FUNCTION_BLOCK FB_Statistic
VAR PERSISTENT
	bSaved:BOOL;
	Data:STRUCT_StatisticsData;
	DataSaved:STRUCT_StatisticsData;
	udiSamplesToSave:UDINT:=500;
	udiSamplesCounter:UDINT:=0;
END_VAR
VAR_INPUT
	bReset:BOOL;
	bRestore:BOOL;
END_VAR
VAR_OUTPUT
	rZScore:REAL;
END_VAR
VAR
	rValue:REAL;
END_VAR

METHOD PRIVATE M_calc_coef
VAR
	rCounter:REAL;
END_VAR
// Check counter and cast to real
IF THIS^.Data.udiCounter=0 THEN
	rCounter:=1;
END_IF
rCounter:=UDINT_TO_REAL(THIS^.Data.udiCounter);
// CALCULATE
// =======================================================
THIS^.Data.rStatCoef:=MAX((1/rCounter),THIS^.Data.rStatCoefMin);
// =======================================================
END_METHOD

METHOD PRIVATE M_calc_dev
VAR
	rRes:REAL;
END_VAR
IF THIS^.Data.rStatCoef=0 OR THIS^.Data.rStatCoef=1 THEN
	THIS^.Data.rDevSum:=0;
ELSE
	IF (THIS^.rValue-THIS^.Data.rMean)=0 THEN
		rRes:=0;
	ELSE
		rRes:=EXPT(THIS^.rValue-THIS^.Data.rMean,2);
	END_IF
	THIS^.Data.rDevSum :=	((1-THIS^.Data.rStatCoef)*THIS^.Data.rDevSum) + 
							(THIS^.Data.rStatCoef*rRes);
END_IF

IF THIS^.Data.rDevSum=0 THEN
	THIS^.Data.rDev:=0;
ELSE
	THIS^.Data.rDev:=SQRT(THIS^.Data.rDevSum);
END_IF
END_METHOD

METHOD PRIVATE M_calc_mean
VAR_INPUT
END_VAR
IF THIS^.Data.rStatCoef=1 THEN
	THIS^.Data.rMean:=THIS^.rValue;
ELSE
	IF THIS^.Data.rStatCoef<>0 THEN
		THIS^.Data.rMean := ((1-THIS^.Data.rStatCoef)*THIS^.Data.rMean) + 
							(THIS^.Data.rStatCoef*THIS^.rValue);
	end_if
END_IF
END_METHOD

METHOD PRIVATE M_calc_min_max
IF THIS^.Data.udiCounter=1 THEN
	THIS^.Data.rMaximum:=THIS^.rValue;
	THIS^.Data.rMinimum:=THIS^.rValue;
END_IF
THIS^.Data.rMinimum:=MIN(THIS^.Data.rMinimum,THIS^.rValue);
THIS^.Data.rMaximum:=MAX(THIS^.Data.rMaximum,THIS^.rValue);
END_METHOD

METHOD M_is_typical : BOOL	// >Return if the current value is in a typical frequence
VAR_INPUT
	freqTypical:REAL;		// Typical frequence
END_VAR
THIS^.rZScore := ABS((THIS^.Data.rMean - THIS^.DataSaved.rMean) / THIS^.DataSaved.rDev);
M_is_typical := THIS^.Data.rMean <= THIS^.DataSaved.rMean- (freqTypical*THIS^.DataSaved.rDev) OR
				THIS^.Data.rMean >= THIS^.DataSaved.rMean+ (freqTypical*THIS^.DataSaved.rDev);
END_METHOD

METHOD PRIVATE M_reset
IF THIS^.bReset THEN
	THIS^.Data.udiCounter:=1;
	THIS^.Data.rStatCoef:=0;
	THIS^.Data.rMinimum:=0;
	THIS^.Data.rMaximum:=0;
	THIS^.Data.rMean:=0;
	THIS^.Data.rDevSum:=0;
	THIS^.Data.rDev:=0;
	THIS^.bSaved:=FALSE;
	THIS^.udiSamplesCounter:=0;
	THIS^.bReset:=FALSE;
END_IF
END_METHOD

METHOD PRIVATE M_restore
VAR_INPUT
END_VAR
IF THIS^.bRestore THEN
	THIS^.Data := THIS^.DataSaved;
	THIS^.bRestore:=FALSE;
END_IF
END_METHOD

METHOD M_run
VAR_INPUT
	rStatCoefMin:REAL;
	rCurrentValue:REAL;
END_VAR
// Reset data
THIS^.M_reset();
// Restore data
THIS^.M_restore();
// Get current data
THIS^.Data.rStatCoefMin:=rStatCoefMin;
THIS^.rValue:=rCurrentValue;
// Calcs
THIS^.M_calc_coef();
THIS^.M_calc_min_max();
THIS^.M_calc_mean();
THIS^.M_calc_dev();
// Save data
THIS^.M_save();
// Update counter
IF THIS^.Data.udiCounter<4294967295 THEN
	THIS^.Data.udiCounter:=THIS^.Data.udiCounter+1;
END_IF
// Update coef counter until coef value if the minumum
IF THIS^.Data.rStatCoefMin<THIS^.Data.rStatCoef THEN
	THIS^.Data.udiCounterCoef:=THIS^.Data.udiCounterCoef+1;
END_IF
END_METHOD

METHOD PRIVATE M_save
IF NOT THIS^.bSaved THEN
	IF THIS^.udiSamplesCounter<THIS^.udiSamplesToSave THEN
		THIS^.udiSamplesCounter:=THIS^.udiSamplesCounter+1;
	ELSE
		THIS^.DataSaved:=THIS^.Data;
		THIS^.bSaved:=TRUE;
		THIS^.udiSamplesCounter:=0;
	END_IF
END_IF
END_METHOD

END_FUNCTION_BLOCK

(* stored: Version 1.1.0.1, ProductVersion 3.1.4024.15
   POU FB_Statistic: Id {f8c8afce-dcce-4abd-ae4d-ed1586048296}, SpecialFunc None
   Folder Calcs: Id {4c417586-d4e3-4952-b697-78d15fa4ce66}
   Method M_calc_coef: Id {3cab2314-2535-45da-9346-cdf0f8f5bd0b}
   Method M_calc_dev: Id {7e7b151d-ffd8-4227-b125-ce70e7a488a1}
   Method M_calc_mean: Id {52ae314d-b209-4612-8880-db6276d84835}
   Method M_calc_min_max: Id {805b42f2-9fbc-4e8d-9a68-902a5847bf79}
   Method M_is_typical: Id {31378273-d22e-493c-a09a-dcf835242b2f}
   Method M_reset: Id {5a4e3e7d-6834-4936-be4a-63521f7e820f}
   Method M_restore: Id {fea33ed9-b3fa-4a8c-b3a7-208c8b903e11}
   Method M_run: Id {3970a310-8d40-4294-ace8-0425422f9804}
   Method M_save: Id {8884862c-a92e-4361-bf2f-df32cf50988a} *)
